TYPE Alarms :
STRUCT
	bIsUsed				: BOOL;
	sName				: STRING; 
	bIsActive			: BOOL;
	bIsAcknowledged		: BOOL;
	uiID				: UINT;
	sAlarmText			: STRING;
	tActiveStartTime	: DT;
	tAcknowlegedTime	: DT;
	uiRepeatCount		: UINT;
	
END_STRUCT
END_TYPE

(* stored: Version 1.1.0.1, ProductVersion 3.1.4024.9
   DUT Alarms: Id {3b1495bb-5bd3-450b-a17b-083265efaee0} *)
